FUNCTION_BLOCK PneumaticInsertion_old
VAR_INPUT
	enable : BOOL;
END_VAR
VAR_OUTPUT
	slider : TeknicEIP;
	screw : AirSlider;
	
	contact : BOOL;
	
	home : BOOL;
	ready : BOOL;
	busy : BOOL;
	error : BOOL;
END_VAR

slider(
	bEnable:= enable, 
	home=> , 
	outerLimit=> , 
	innerLimit=> , 
	done=> , 
	contact=> contact, 
	homeSet=> );
	
screw(
	bEnable:= enable, 
	direction=> , 
	valveIn=> , 
	valveOut=> , 
	contact=> , 
	home=> , 
	innerLimit=> , 
	ready=> , 
	busy=> , 
	error=> , 
	homeSet=> );

home := screw.home AND slider.home;
busy := slider.busy OR screw.busy;
error := slider.error OR screw.error;

METHOD align : BOOL
VAR_INPUT
	targetPos : REAL;
END_VAR
IF slider.position < targetPos THEN
	slider.traverse(direction := TRUE);
	
ELSIF slider.position > targetPos THEN
	slider.traverse(direction := FALSE);
	
ELSE
	align := TRUE;
	
END_IF
END_METHOD

METHOD homingSequence : BOOL
IF NOT screw.homeSet THEN
	screw.homingSequence();
END_IF

IF NOT slider.homeSet THEN
	slider.homingSequence();
END_IF

homingSequence := screw.homeSet AND slider.homeSet;
END_METHOD

METHOD press : BOOL
VAR_INPUT
	//direction : BOOL; //direction (F = inwards, T = outwards)
	//distance : DINT;
END_VAR
slider.traverse(direction := FALSE);
END_METHOD

METHOD release : BOOL
VAR_INPUT
END_VAR
slider.traverse(direction := TRUE);
END_METHOD

METHOD slideContinuous : BOOL
VAR_INPUT
	direction : BOOL; //T = positive direction, F = negative direction
END_VAR
slider.traverse(direction := direction);
END_METHOD

END_FUNCTION_BLOCK

(* stored: Version 1.1.0.1, ProductVersion 3.1.4024.11
   POU PneumaticInsertion_old: Id {b81c5df3-3bac-4f9d-9b77-7bbeccd1dc76}, SpecialFunc None
   Method align: Id {89be0205-36be-4635-bf1d-734fb40c3796}
   Method homingSequence: Id {d7cd42ba-bf91-49d9-b290-abbbea3d3ad6}
   Method press: Id {b1e47417-f59e-4f47-a453-5b14f0c0ab9e}
   Method release: Id {6735797f-0df0-46da-8234-935ba24cde58}
   Method slideContinuous: Id {b7ff75db-864c-438f-bfb9-1fb8fcf5dcaf} *)
